# EPICS substitutions: src/makeBaseApp/top/archiver/_IOC_.substitutions
# Archiver request file
## Replace _IOCPVROOT_ with the PV prefix used for
## iocAdmin PV's on this IOC
file "iocAdmin.arch_template"
{
	{ IOC = "_IOCPVROOT_" }
}
